(* Logix 5000 project; controller WWTP_SOLIDS_CLX vendor 1 type 14 code 54 rev 17.2; software revision 17.00; part 7 of 16 *)
(* tags used below, declared in another part *)
   Inp_PVBad : BOOL;   // 1=Scale PV or I/O Quality Bad, 0=OK
   Inp_PVUncertain : BOOL;   // 1=Scale PV Quality Uncertain, 0=OK
   Inp_CtrldEqpFault : BOOL;   // Controlled Equipment device or I/O status 0=OK, 1=fail
   Inp_Sim : BOOL;   // 1=Simulate working weigh scale; 0=use actual weight input
   Cfg_HasDribble : BOOL;   // 1=Slow to Dribble before complete, 0=use complete only
   Cfg_PCmdClear : BOOL;   // 1=Clear Program Commands on receipt 0=Leave Set
   Cfg_HasOverTolAlm : BOOL;   // 1=Over Tolerance Alarm exists and will be checked
   Cfg_HasUnderTolAlm : BOOL;   // 1=Under Tolerance Alarm exists and will be checked
   Cfg_HasTareFaultAlm : BOOL;   // 1=Tare Fault Alarm exists and will be checked
   Cfg_HasEqpFaultAlm : BOOL;   // 1=Equipment Fault Alarm exists and will be checked
   Cfg_OverTolResetReqd : BOOL;   // 1=Reset requied to clear Out of Tolerance High Alarm
   Cfg_UnderTolResetReqd : BOOL;   // 1=Reset required to clear Out of Tolerance Low Alarm
   Cfg_TareFaultResetReqd : BOOL;   // 1=Reset required to clear Tare Fault Alarm
   Cfg_EqpFaultResetReqd : BOOL;   // 1=Reset required to clear Equipment Fault Alarm
   Cfg_OverTolAckReqd : BOOL;   // 1=Acknowledge required for Out of Tolerance High Alarm
   Cfg_UnderTolAckReqd : BOOL;   // 1=Acknowledge required for Out of Tolerance Low Alarm
   Cfg_TareFaultAckReqd : BOOL;   // 1=Acknowledge required for Tare Fault Alarm
   Cfg_EqpFaultAckReqd : BOOL;   // 1=Acknowledge required for Equipment Fault Alarm
   Cfg_OverTolSeverity : SINT;   // Over Tolerance Alarm Severity 1=info, 2=warn, 3=excep, 4=fault
   Cfg_UnderTolSeverity : SINT;   // Under Tolerance Alarm Severity 1=info, 2=warn, 3=excep, 4=fault
   Cfg_TareFaultSeverity : SINT;   // Tare Fault Alarm Severity 1=info, 2=warn, 3=excep, 4=fault
   Cfg_EqpFaultSeverity : SINT;   // Equipment Fault Alarm Severity 1=info, 2=warn, 3=excep, 4=fault
   Cfg_InpRawMin : REAL;   // Minimum unscaled weight input
   Cfg_InpRawMax : REAL;   // Maximum unscaled weight input
   Cfg_PVEUMin : REAL;   // Minimum scaled weight PV input (EU)
   Cfg_PVEUMax : REAL;   // Maximum scaled weight PV input (EU)
   Cfg_MaxQty : REAL;   // Maximum allowed quantity to deliver (setpoint) (EU)
   Cfg_RateTime : REAL;   // Time factor for rate (60 for /min, 3600 for /hr) (Sec)
   Cfg_RateFiltTC : REAL;   // Filter Time Constant (sec) for calculated Rate
   Cfg_TareFaultLim : REAL;   // Amount (EU) scale can drift after Tare before starting flow without Faulting
   Cfg_SimStartWt : REAL;   // Weight to start from (tare to) in simulation (EU)
   Cfg_SimRate : REAL;   // Rate at which to deliver when running in Simulation (EU/rate time)
   Cfg_SimDribbleRate : REAL;   // Rate at which to dribble when running in Simulation (EU/rate time)
   PCmd_OverTolAck : BOOL;   // Program Command to Acknowledge Out of Tolerance High Alarm
   PCmd_OverTolInhibit : BOOL;   // Program Command to Inhibit Out of Tolerance High Alarm
   PCmd_OverTolUninhibit : BOOL;   // Program Command to Uninhibit Out of Tolerance High Alarm
   PCmd_UnderTolAck : BOOL;   // Program Command to Acknowledge Out of Tolerance Low Alarm
   PCmd_UnderTolInhibit : BOOL;   // Program Command to Inhibit Out of Tolerance Low Alarm
   PCmd_UnderTolUninhibit : BOOL;   // Program Command to Uninhibit Out of Tolerance Low Alarm
   PCmd_TareFaultAck : BOOL;   // Program Command to Acknowledge Tare Fault Alarm
   PCmd_TareFaultInhibit : BOOL;   // Program Command to Inhibit Tare Fault Alarm
   PCmd_TareFaultUninhibit : BOOL;   // Program Command to Uninhibit Tare Fault Alarm
   PCmd_EqpFaultAck : BOOL;   // Program Command to Acknowledge Equipment Fault Alarm
   PCmd_EqpFaultInhibit : BOOL;   // Program Command to Inhibit Equipment Fault Alarm
   PCmd_EqpFaultUninhibit : BOOL;   // Program Command to Uninhibit Equipment Fault Alarm
   Out_RunFlow : BOOL;   // 1=Deliver at Full (fast) Flow
   Out_DribbleFlow : BOOL;   // 1=Deliver at Dribble (slow) Flow
   Out_StopFlow : BOOL;   // 1=Stop Delivery Equipment
   Val_Qty : REAL;   // Quantity actually delivered (totalizer output) (EU)
   Val_SP : REAL;   // Amount to be delivered (Setpoint) (EU)
   Val_PctComplete : REAL;   // Percent Complete (for Progress Bar on HMI) 0.0 to 100.0%
   Val_DribbleQty : REAL;   // Amount to be delivered at slow rate (EU)
   Val_Preact : REAL;   // Amount before SP at which flow will be stopped (EU)
   Val_PVEUMin : REAL;   // Minimum of scaled range = MIN (Cfg_PVEUMin, Cfg_PVEUMax)
   Val_PVEUMax : REAL;   // Maximum of scaled range = MAX (Cfg_PVEUMin, Cfg_PVEUMax)
   Val_Notify : SINT;   // Current Alarm Level and Acknowledgement (enumeration)
   Sts_Tared : BOOL;   // Scale Tare completed, Qty = 0.0
   Sts_FlowRunning : BOOL;   // 1=Flow is Running (Out_Run is ON)
   Sts_FlowDribble : BOOL;   // 1=Flow is slowed to Dribble (Out_Dribble is ON)
   Sts_FlowStopped : BOOL;   // 1=Flow is Stopped (Out_Stop is ON)
   Sts_Bumping : BOOL;   // 1=Bump flow (timed) is active
   Sts_Complete : BOOL;   // 1=Total Delivered > (SP - Preact)
   Sts_Available : BOOL;   // 1=Dosing available for control by automation (Prog)
   Sts_PVBad : BOOL;   // 1=Weight PV and Rate PV Quality Bad (I/O fail), 0=OK
   Sts_PVUncertain : BOOL;   // 1=Weight PV and Rate PV Quality is Uncertian, 0=OK
   Sts_Err : BOOL;   // 1=Error: Bad Configuration, see detail Err bits for reason
   Err_Raw : BOOL;   // 1=Error: Cfg_InpRawMax or Cfg_InpRawMin invalid
   Err_EU : BOOL;   // 1=Error: Cfg_PVEUMax or Cfg_PVEUMin invalid
   Err_Rate : BOOL;   // 1=Error: Cfg_RateFiltTC or Cfg_RateTime invalid
   Err_Limit : BOOL;   // 1=Error: Cfg_MaxQty invalid
   Err_Sim : BOOL;   // 1=Error: Cfg_SimDribbleRate or Cfg_SimRate invalid
   Err_Timer : BOOL;   // 1=Error: Cfg_BumpT (use 0.0 to 2147483.647)
   Err_Alarm : BOOL;   // 1=Error: Alarm Min Duration or Severity Cfg Invalid
   Sts_Maint : BOOL;   // 1=Mode is Maintenance (supersedes Prog, Oper)
   Sts_Prog : BOOL;   // 1=Mode is Program (auto)
   Sts_Oper : BOOL;   // 1=Mode is Operator (manual)
   Sts_ProgOperLock : BOOL;   // 1=Program or Operator has requested Mode Lock
   Sts_OverTol : BOOL;   // 1=Delivery Out of Tolerance High
   Alm_OverTol : BOOL;   // 1=Delivery Out of Tolerance High Alarm
   Ack_OverTol : BOOL;   // 1=Out of Tolerance High Alarm has been acknowledged
   Sts_OverTolDisabled : BOOL;   // 1=Out of Tolerance High Alarm has been disabled (will not be sent)
   Sts_OverTolInhibited : BOOL;   // 1=Out of Tolerance High Alarm has been inhibited by logic
   Sts_OverTolSuppressed : BOOL;   // 1=Out of Tolerance High Alarm has been suppressed (logged only)
   Sts_UnderTol : BOOL;   // 1=Delivery Out of Tolerance Low
   Alm_UnderTol : BOOL;   // 1=Delivery Out of Tolerance Low Alarm
   Ack_UnderTol : BOOL;   // 1=Out of Tolerance Low Alarm has been acknowledged
   Sts_UnderTolDisabled : BOOL;   // 1=Out of Tolerance Low Alarm has been disabled (will not be sent)
   Sts_UnderTolInhibited : BOOL;   // 1=Out of Tolerance Low Alarm has been inhibited by logic
   Sts_UnderTolSuppressed : BOOL;   // 1=Out of Tolerance Low Alarm has been suppressed (logged only)
   Sts_TareFault : BOOL;   // 1=Scale reading moved unexpectedly since Tare
   Alm_TareFault : BOOL;   // 1=Warning: scale reading moved since Tare
   Ack_TareFault : BOOL;   // 1=Tare Fault Alarm has been acknowledged
   Sts_TareFaultDisabled : BOOL;   // 1=Tare Fault Alarm is Disabled (not saved or sent)
   Sts_TareFaultInhibited : BOOL;   // 1=Tare Fault Alarm has been inhibited by logic
   Sts_TareFaultSuppressed : BOOL;   // 1=Tare Fault Alarm has been suppressed (logged only)
   Sts_EqpFault : BOOL;   // 1=Equipment Fault Detected
   Alm_EqpFault : BOOL;   // 1=Equipment Fault Alarm
   Ack_EqpFault : BOOL;   // 1=Equipment Fault Alarm has been acknowledged
   Sts_EqpFaultDisabled : BOOL;   // 1=Equipment Fault Alarm is Disabled (not saved or sent)
   Sts_EqpFaultInhibited : BOOL;   // 1=Equipment Fault Alarm has been inhibited by logic
   Sts_EqpFaultSuppressed : BOOL;   // 1=Equipment Fault Alarm has been suppressed (logged only)
   Rdy_Tare : BOOL;   // 1=Ready for OCmd_Tare (enables button)
   Rdy_StartFlow : BOOL;   // 1=Ready for OCmd_StartFlow (enables button)
   Rdy_StopFlow : BOOL;   // 1=Ready for OCmd_StopFlow (enables button)
   Rdy_CheckTol : BOOL;   // 1-Ready for OCmd_CheckTol (enables button)
   Rdy_Bump : BOOL;   // 1=Ready for OCmd_Bump (enables button)
   Rdy_Reset : BOOL;   // 1=Ready for OCmd_Reset (enables button)
   Wrk_Notify : DINT;   // Buffer for building Val_Notify
   Mode : P_Mode;   // Analog Input Mode Selection
   Wrk_Tare : BOOL;   // Request to Tare Scale received
   TareFault : P_Alarm;   // Scale not holding at point at which Tared Alarm
   UnderTol : P_Alarm;   // Final Quantity Below Low Tolerance Alarm
   OverTol : P_Alarm;   // Final Quantity Above High Tolerance Alarm
   EqpFault : P_Alarm;   // Equipment (Sensor, Controlled Equip.) Fault Alarm
   Wrk_RunFlow : BOOL;   // 1=Flow (full)( should be running
   Wrk_BumpFlow : BOOL;   // Operator requested bump flow to make up Under Tolerance
   Wrk_BumpT : TIMER;   // Bump Timer for shot of flow to make up Under Tolerance
   Wrk_PctComplete : REAL;   // Percent Complete calculation intermediate
   Wrk_InpInfNaN : BOOL;   // Input Weight is Infinite or NaN
(* P_DoseWS, continued *)

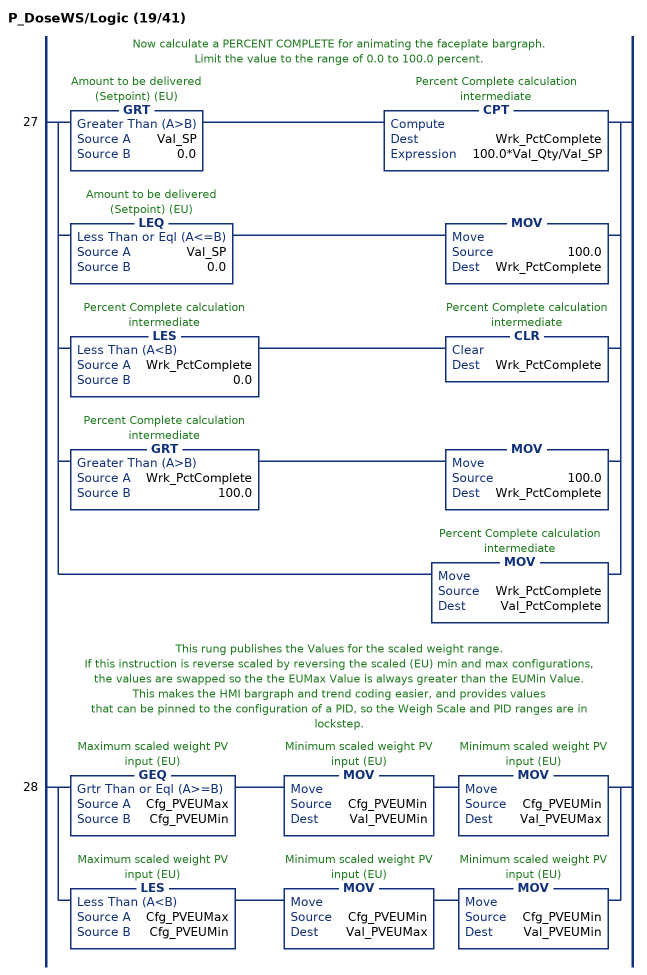
   [picture p136: P_DoseWS/Logic rungs 27-28]
   // Now calculate a PERCENT COMPLETE for animating the faceplate bargraph.
   // Limit the value to the range of 0.0 to 100.0 percent.
   27: [GRT(Val_SP,0.0) CPT(Wrk_PctComplete,100.0*Val_Qty/Val_SP) ,LEQ(Val_SP,0.0) MOV(100.0,Wrk_PctComplete) ,LES(Wrk_PctComplete,0.0) CLR(Wrk_PctComplete) ,GRT(Wrk_PctComplete,100.0) MOV(100.0,Wrk_PctComplete) ,MOV(Wrk_PctComplete,Val_PctComplete) ];
   // This rung publishes the Values for the scaled weight range.
   // If this instruction is reverse scaled by reversing the scaled (EU) min and max configurations,
   // the values are swapped so the the EUMax Value is always greater than the EUMin Value.
   // This makes the HMI bargraph and trend coding easier, and provides values
   // that can be pinned to the configuration of a PID, so the Weigh Scale and PID ranges are in lockstep.
   28: [GEQ(Cfg_PVEUMax,Cfg_PVEUMin) MOV(Cfg_PVEUMin,Val_PVEUMin) MOV(Cfg_PVEUMin,Val_PVEUMax) ,LES(Cfg_PVEUMax,Cfg_PVEUMin) MOV(Cfg_PVEUMin,Val_PVEUMax) MOV(Cfg_PVEUMin,Val_PVEUMin) ];
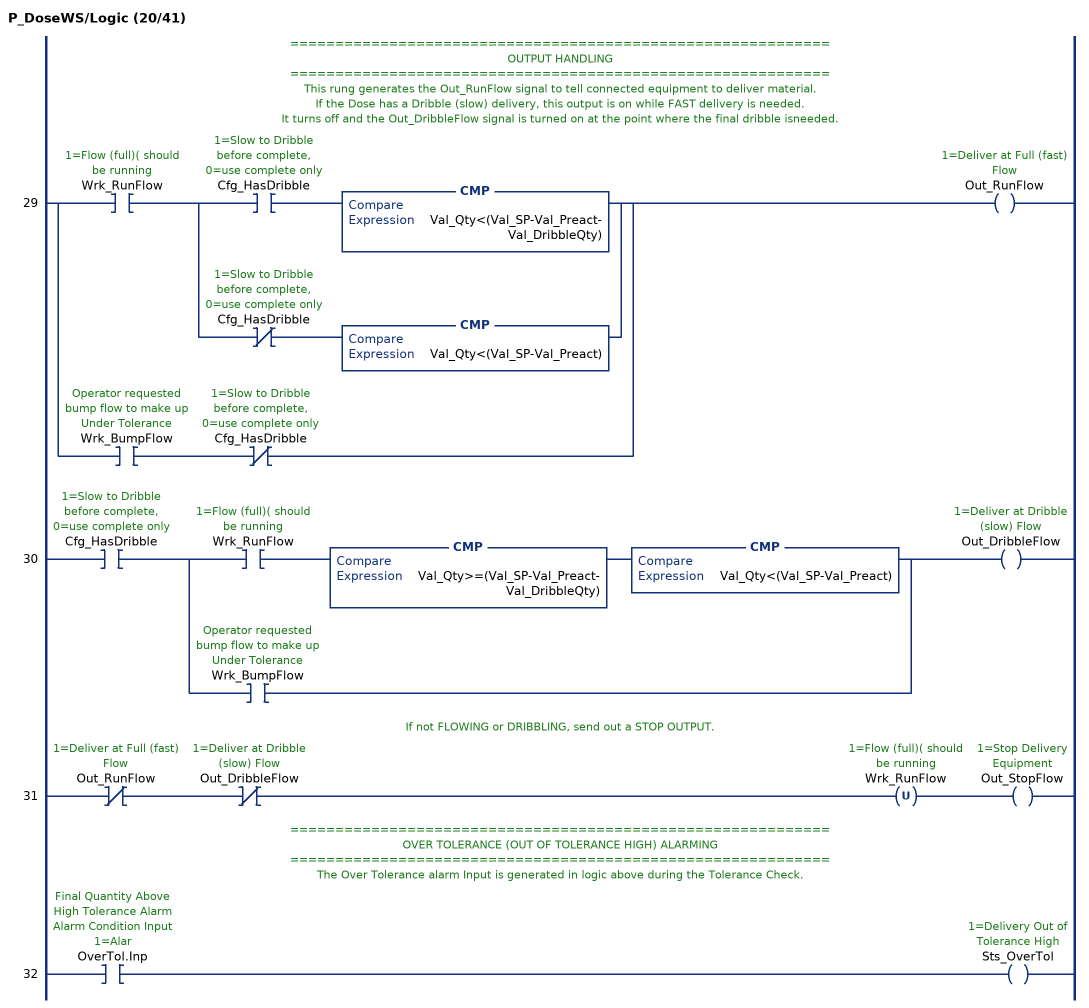
   // ============================================================
   // OUTPUT HANDLING
   // ============================================================
   // This rung generates the Out_RunFlow signal to tell connected equipment to deliver material.
   // If the Dose has a Dribble (slow) delivery, this output is on while FAST delivery is needed.
   // It turns off and the Out_DribbleFlow signal is turned on at the point where the final dribble isneeded.
   29: [XIC(Wrk_RunFlow) [XIC(Cfg_HasDribble) CMP(Val_Qty<(Val_SP-Val_Preact-Val_DribbleQty)) ,XIO(Cfg_HasDribble) CMP(Val_Qty<(Val_SP-Val_Preact)) ] ,XIC(Wrk_BumpFlow) XIO(Cfg_HasDribble) ]OTE(Out_RunFlow);
   30: XIC(Cfg_HasDribble)[XIC(Wrk_RunFlow) CMP(Val_Qty>=(Val_SP-Val_Preact-Val_DribbleQty)) CMP(Val_Qty<(Val_SP-Val_Preact)) ,XIC(Wrk_BumpFlow) ]OTE(Out_DribbleFlow);
   // If not FLOWING or DRIBBLING, send out a STOP OUTPUT.
   31: XIO(Out_RunFlow)XIO(Out_DribbleFlow)OTU(Wrk_RunFlow)OTE(Out_StopFlow);
   // ============================================================
   // OVER TOLERANCE (OUT OF TOLERANCE HIGH) ALARMING
   // ============================================================
   // The Over Tolerance alarm Input is generated in logic above during the Tolerance Check.
   32: XIC(OverTol.Inp)OTE(Sts_OverTol);
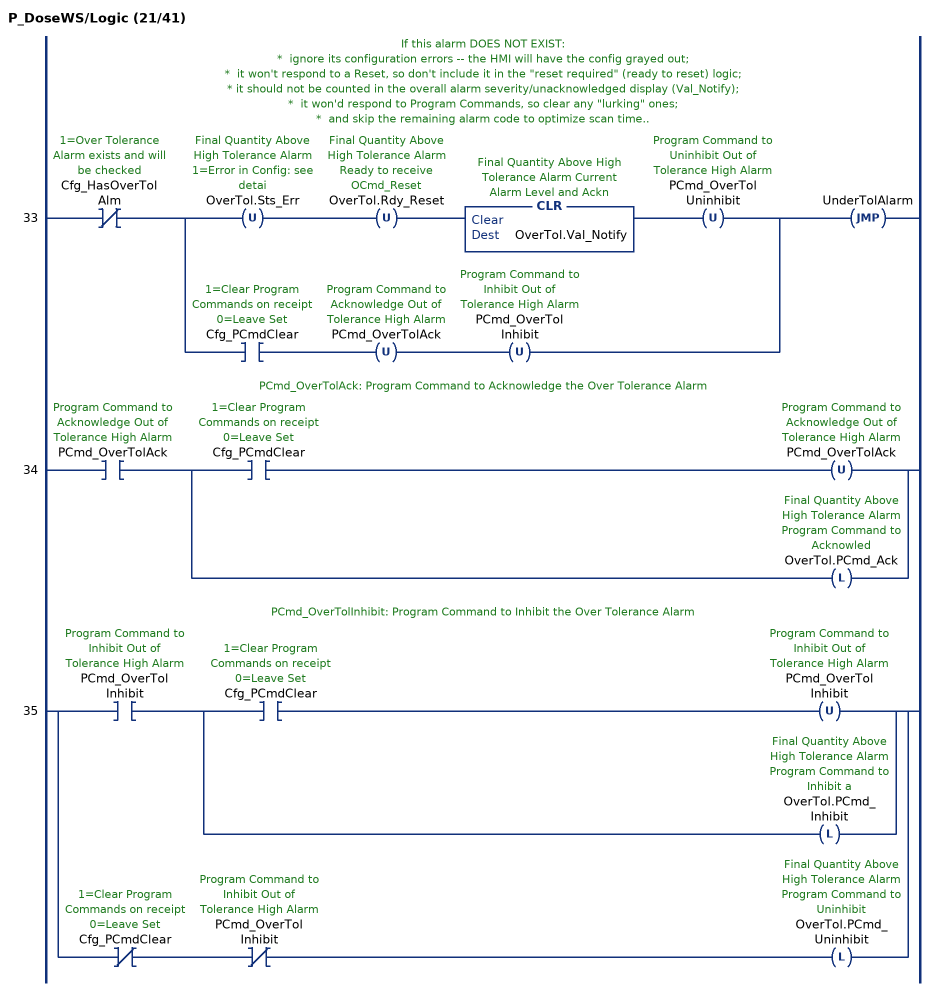
   // If this alarm DOES NOT EXIST:
   // *  ignore its configuration errors -- the HMI will have the config grayed out;
   // *  it won't respond to a Reset, so don't include it in the "reset required" (ready to reset) logic;
   // * it should not be counted in the overall alarm severity/unacknowledged display (Val_Notify);
   // *  it won'd respond to Program Commands, so clear any "lurking" ones;
   // *  and skip the remaining alarm code to optimize scan time..
   33: XIO(Cfg_HasOverTolAlm)[OTU(OverTol.Sts_Err) OTU(OverTol.Rdy_Reset) CLR(OverTol.Val_Notify) OTU(PCmd_OverTolUninhibit) ,XIC(Cfg_PCmdClear) OTU(PCmd_OverTolAck) OTU(PCmd_OverTolInhibit) ]JMP(UnderTolAlarm);
   // PCmd_OverTolAck: Program Command to Acknowledge the Over Tolerance Alarm
   34: XIC(PCmd_OverTolAck)[XIC(Cfg_PCmdClear) OTU(PCmd_OverTolAck) ,OTL(OverTol.PCmd_Ack) ];
   // PCmd_OverTolInhibit: Program Command to Inhibit the Over Tolerance Alarm
   35: [XIC(PCmd_OverTolInhibit) [XIC(Cfg_PCmdClear) OTU(PCmd_OverTolInhibit) ,OTL(OverTol.PCmd_Inhibit) ] ,XIO(Cfg_PCmdClear) XIO(PCmd_OverTolInhibit) OTL(OverTol.PCmd_Uninhibit) ];
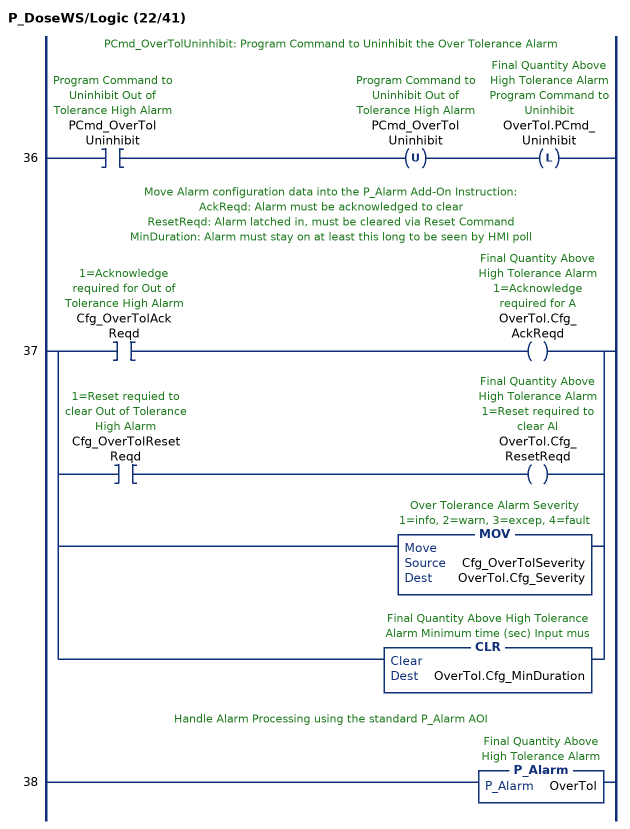
   // PCmd_OverTolUninhibit: Program Command to Uninhibit the Over Tolerance Alarm
   36: XIC(PCmd_OverTolUninhibit)OTU(PCmd_OverTolUninhibit)OTL(OverTol.PCmd_Uninhibit);
   // Move Alarm configuration data into the P_Alarm Add-On Instruction:
   // AckReqd: Alarm must be acknowledged to clear
   // ResetReqd: Alarm latched in, must be cleared via Reset Command
   // MinDuration: Alarm must stay on at least this long to be seen by HMI poll
   37: [XIC(Cfg_OverTolAckReqd) OTE(OverTol.Cfg_AckReqd) ,XIC(Cfg_OverTolResetReqd) OTE(OverTol.Cfg_ResetReqd) ,MOV(Cfg_OverTolSeverity,OverTol.Cfg_Severity) ,CLR(OverTol.Cfg_MinDuration) ];
   // Handle Alarm Processing using the standard P_Alarm AOI
   38: P_Alarm(OverTol);
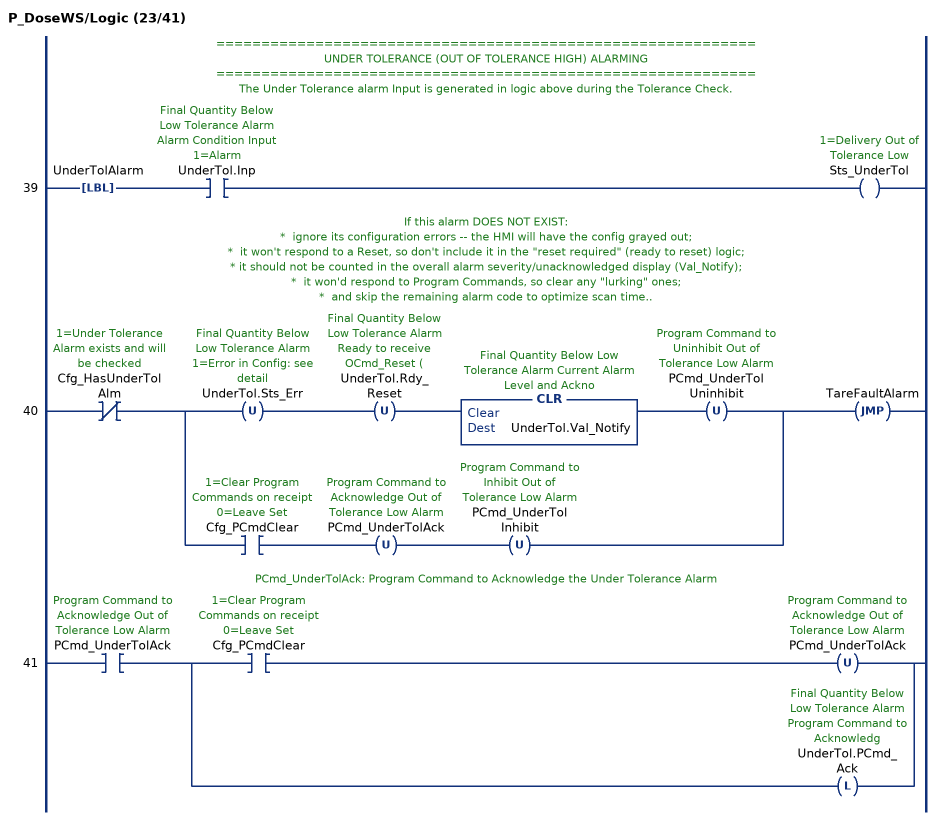
   // ============================================================
   // UNDER TOLERANCE (OUT OF TOLERANCE HIGH) ALARMING
   // ============================================================
   // The Under Tolerance alarm Input is generated in logic above during the Tolerance Check.
   39: LBL(UnderTolAlarm)XIC(UnderTol.Inp)OTE(Sts_UnderTol);
   // If this alarm DOES NOT EXIST:
   // *  ignore its configuration errors -- the HMI will have the config grayed out;
   // *  it won't respond to a Reset, so don't include it in the "reset required" (ready to reset) logic;
   // * it should not be counted in the overall alarm severity/unacknowledged display (Val_Notify);
   // *  it won'd respond to Program Commands, so clear any "lurking" ones;
   // *  and skip the remaining alarm code to optimize scan time..
   40: XIO(Cfg_HasUnderTolAlm)[OTU(UnderTol.Sts_Err) OTU(UnderTol.Rdy_Reset) CLR(UnderTol.Val_Notify) OTU(PCmd_UnderTolUninhibit) ,XIC(Cfg_PCmdClear) OTU(PCmd_UnderTolAck) OTU(PCmd_UnderTolInhibit) ]JMP(TareFaultAlarm);
   // PCmd_UnderTolAck: Program Command to Acknowledge the Under Tolerance Alarm
   41: XIC(PCmd_UnderTolAck)[XIC(Cfg_PCmdClear) OTU(PCmd_UnderTolAck) ,OTL(UnderTol.PCmd_Ack) ];
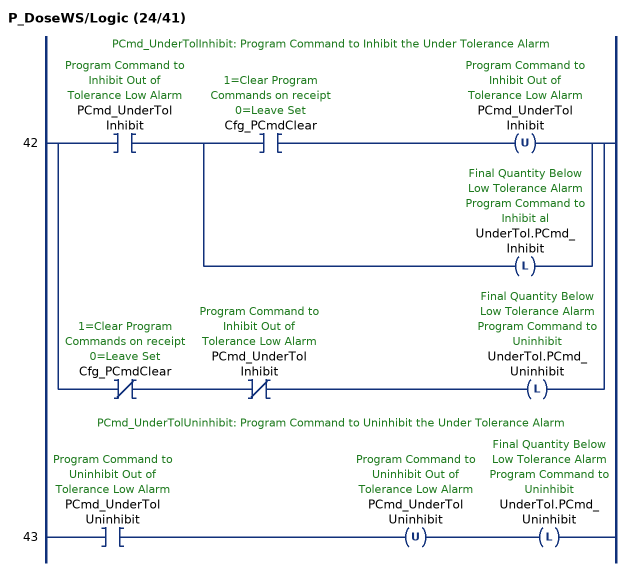
   // PCmd_UnderTolInhibit: Program Command to Inhibit the Under Tolerance Alarm
   42: [XIC(PCmd_UnderTolInhibit) [XIC(Cfg_PCmdClear) OTU(PCmd_UnderTolInhibit) ,OTL(UnderTol.PCmd_Inhibit) ] ,XIO(Cfg_PCmdClear) XIO(PCmd_UnderTolInhibit) OTL(UnderTol.PCmd_Uninhibit) ];
   // PCmd_UnderTolUninhibit: Program Command to Uninhibit the Under Tolerance Alarm
   43: XIC(PCmd_UnderTolUninhibit)OTU(PCmd_UnderTolUninhibit)OTL(UnderTol.PCmd_Uninhibit);
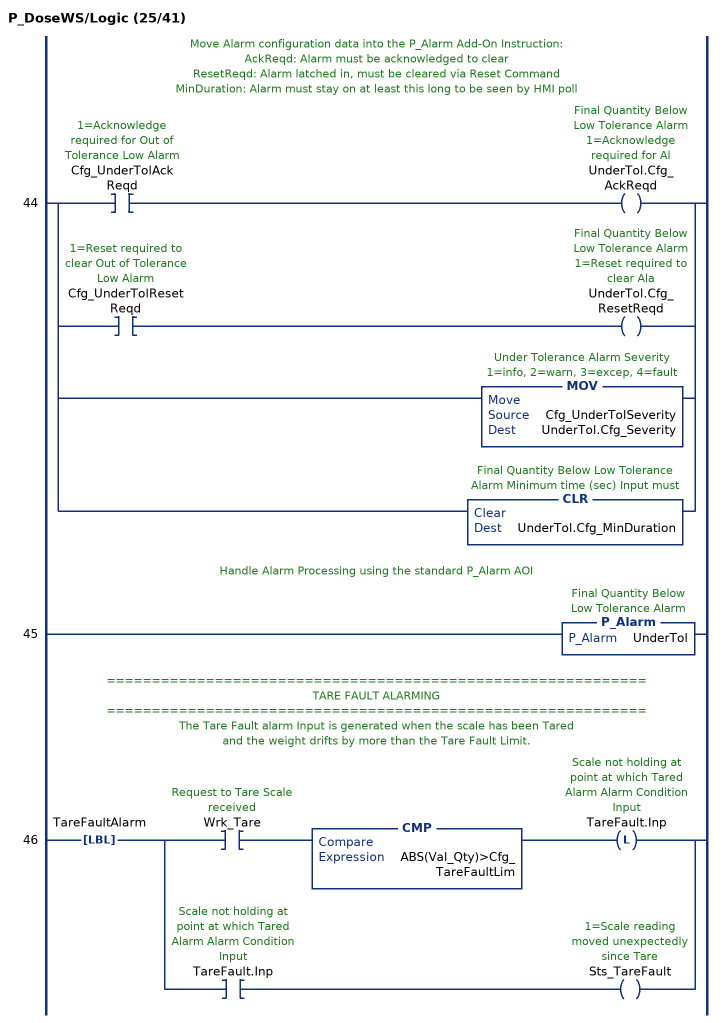
   // Move Alarm configuration data into the P_Alarm Add-On Instruction:
   // AckReqd: Alarm must be acknowledged to clear
   // ResetReqd: Alarm latched in, must be cleared via Reset Command
   // MinDuration: Alarm must stay on at least this long to be seen by HMI poll
   44: [XIC(Cfg_UnderTolAckReqd) OTE(UnderTol.Cfg_AckReqd) ,XIC(Cfg_UnderTolResetReqd) OTE(UnderTol.Cfg_ResetReqd) ,MOV(Cfg_UnderTolSeverity,UnderTol.Cfg_Severity) ,CLR(UnderTol.Cfg_MinDuration) ];
   // Handle Alarm Processing using the standard P_Alarm AOI
   45: P_Alarm(UnderTol);
   // ============================================================
   // TARE FAULT ALARMING
   // ============================================================
   // The Tare Fault alarm Input is generated when the scale has been Tared
   // and the weight drifts by more than the Tare Fault Limit.
   46: LBL(TareFaultAlarm)[XIC(Wrk_Tare) CMP(ABS(Val_Qty)>Cfg_TareFaultLim) OTL(TareFault.Inp) ,XIC(TareFault.Inp) OTE(Sts_TareFault) ];
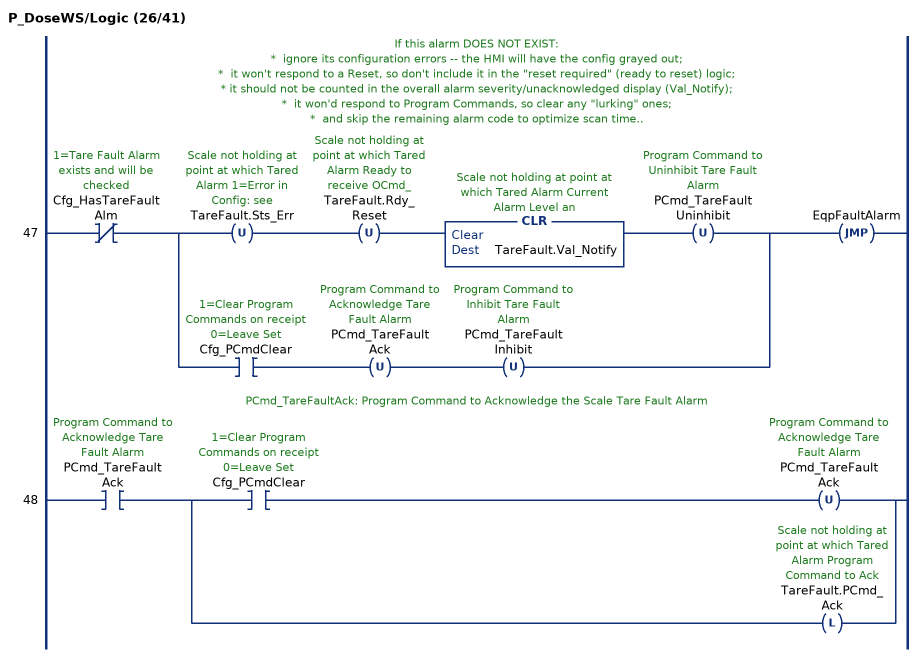
   // If this alarm DOES NOT EXIST:
   // *  ignore its configuration errors -- the HMI will have the config grayed out;
   // *  it won't respond to a Reset, so don't include it in the "reset required" (ready to reset) logic;
   // * it should not be counted in the overall alarm severity/unacknowledged display (Val_Notify);
   // *  it won'd respond to Program Commands, so clear any "lurking" ones;
   // *  and skip the remaining alarm code to optimize scan time..
   47: XIO(Cfg_HasTareFaultAlm)[OTU(TareFault.Sts_Err) OTU(TareFault.Rdy_Reset) CLR(TareFault.Val_Notify) OTU(PCmd_TareFaultUninhibit) ,XIC(Cfg_PCmdClear) OTU(PCmd_TareFaultAck) OTU(PCmd_TareFaultInhibit) ]JMP(EqpFaultAlarm);
   // PCmd_TareFaultAck: Program Command to Acknowledge the Scale Tare Fault Alarm
   48: XIC(PCmd_TareFaultAck)[XIC(Cfg_PCmdClear) OTU(PCmd_TareFaultAck) ,OTL(TareFault.PCmd_Ack) ];
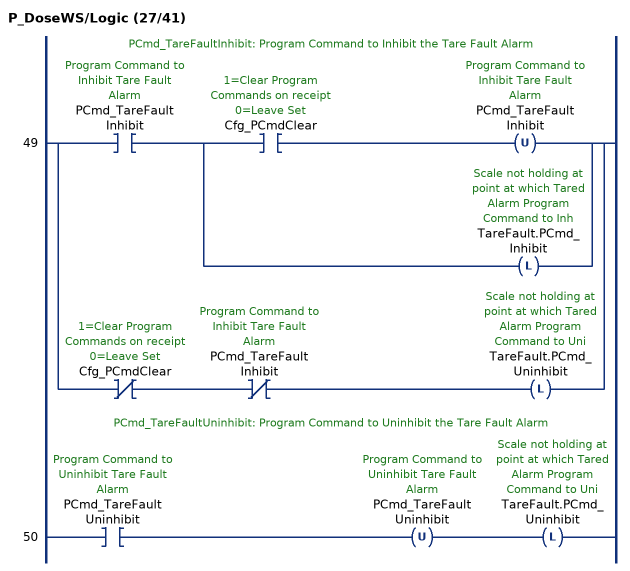
   // PCmd_TareFaultInhibit: Program Command to Inhibit the Tare Fault Alarm
   49: [XIC(PCmd_TareFaultInhibit) [XIC(Cfg_PCmdClear) OTU(PCmd_TareFaultInhibit) ,OTL(TareFault.PCmd_Inhibit) ] ,XIO(Cfg_PCmdClear) XIO(PCmd_TareFaultInhibit) OTL(TareFault.PCmd_Uninhibit) ];
   // PCmd_TareFaultUninhibit: Program Command to Uninhibit the Tare Fault Alarm
   50: XIC(PCmd_TareFaultUninhibit)OTU(PCmd_TareFaultUninhibit)OTL(TareFault.PCmd_Uninhibit);
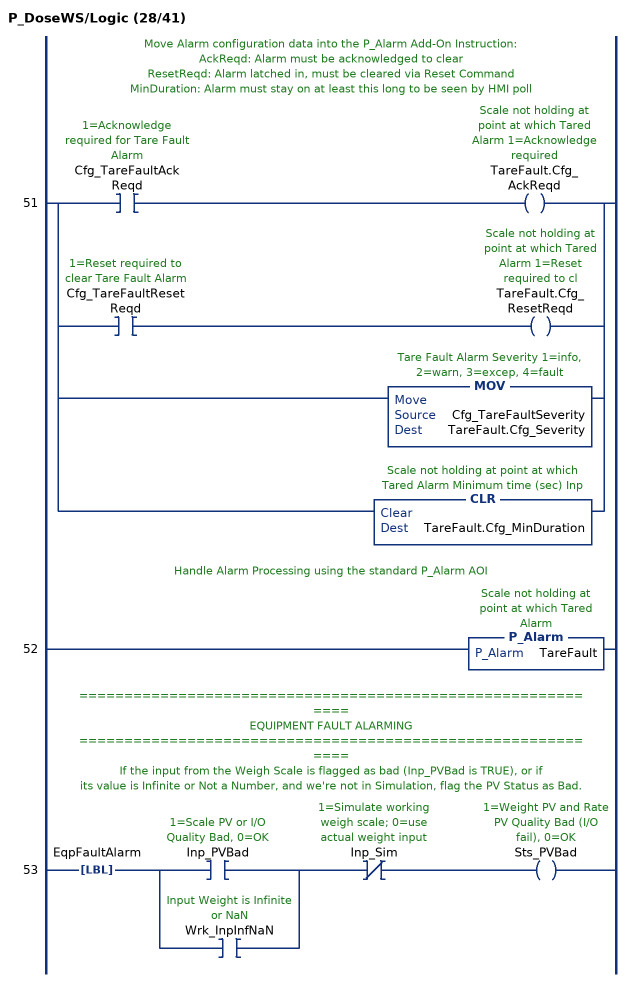
   // Move Alarm configuration data into the P_Alarm Add-On Instruction:
   // AckReqd: Alarm must be acknowledged to clear
   // ResetReqd: Alarm latched in, must be cleared via Reset Command
   // MinDuration: Alarm must stay on at least this long to be seen by HMI poll
   51: [XIC(Cfg_TareFaultAckReqd) OTE(TareFault.Cfg_AckReqd) ,XIC(Cfg_TareFaultResetReqd) OTE(TareFault.Cfg_ResetReqd) ,MOV(Cfg_TareFaultSeverity,TareFault.Cfg_Severity) ,CLR(TareFault.Cfg_MinDuration) ];
   // Handle Alarm Processing using the standard P_Alarm AOI
   52: P_Alarm(TareFault);
   // ============================================================
   // EQUIPMENT FAULT ALARMING
   // ============================================================
   // If the input from the Weigh Scale is flagged as bad (Inp_PVBad is TRUE), or if
   // its value is Infinite or Not a Number, and we're not in Simulation, flag the PV Status as Bad.
   53: LBL(EqpFaultAlarm)[XIC(Inp_PVBad) ,XIC(Wrk_InpInfNaN) ]XIO(Inp_Sim)OTE(Sts_PVBad);
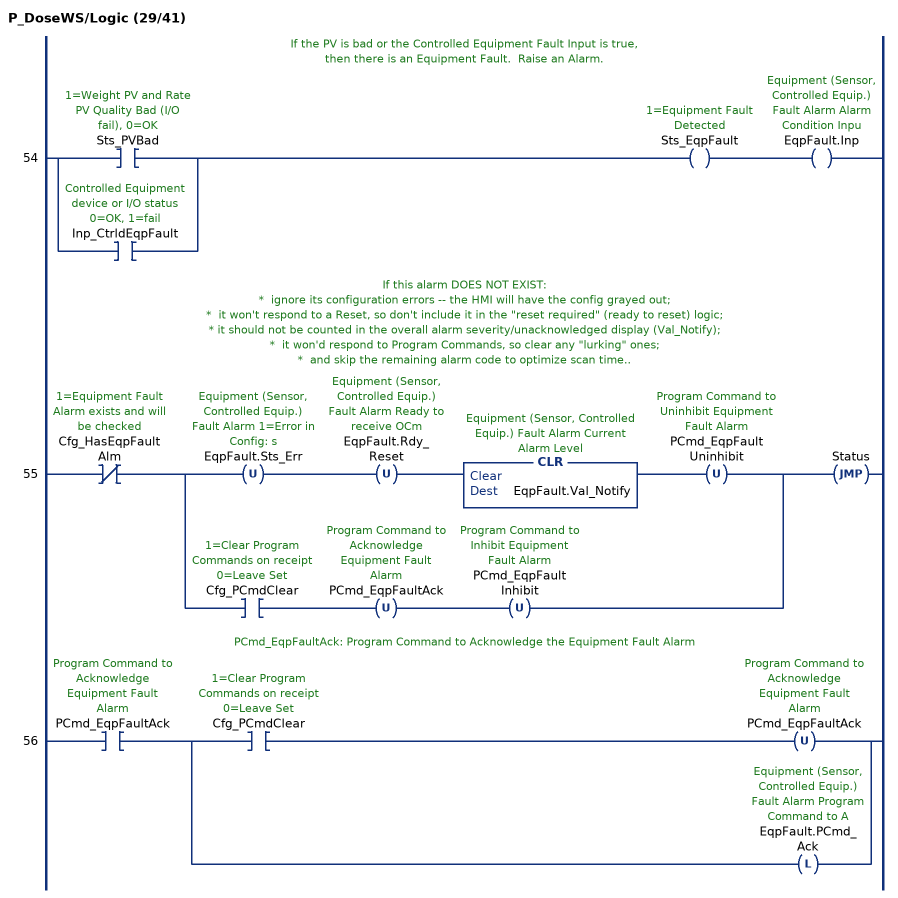
   // If the PV is bad or the Controlled Equipment Fault Input is true,
   // then there is an Equipment Fault.  Raise an Alarm.
   54: [XIC(Sts_PVBad) ,XIC(Inp_CtrldEqpFault) ]OTE(Sts_EqpFault)OTE(EqpFault.Inp);
   // If this alarm DOES NOT EXIST:
   // *  ignore its configuration errors -- the HMI will have the config grayed out;
   // *  it won't respond to a Reset, so don't include it in the "reset required" (ready to reset) logic;
   // * it should not be counted in the overall alarm severity/unacknowledged display (Val_Notify);
   // *  it won'd respond to Program Commands, so clear any "lurking" ones;
   // *  and skip the remaining alarm code to optimize scan time..
   55: XIO(Cfg_HasEqpFaultAlm)[OTU(EqpFault.Sts_Err) OTU(EqpFault.Rdy_Reset) CLR(EqpFault.Val_Notify) OTU(PCmd_EqpFaultUninhibit) ,XIC(Cfg_PCmdClear) OTU(PCmd_EqpFaultAck) OTU(PCmd_EqpFaultInhibit) ]JMP(Status);
   // PCmd_EqpFaultAck: Program Command to Acknowledge the Equipment Fault Alarm
   56: XIC(PCmd_EqpFaultAck)[XIC(Cfg_PCmdClear) OTU(PCmd_EqpFaultAck) ,OTL(EqpFault.PCmd_Ack) ];
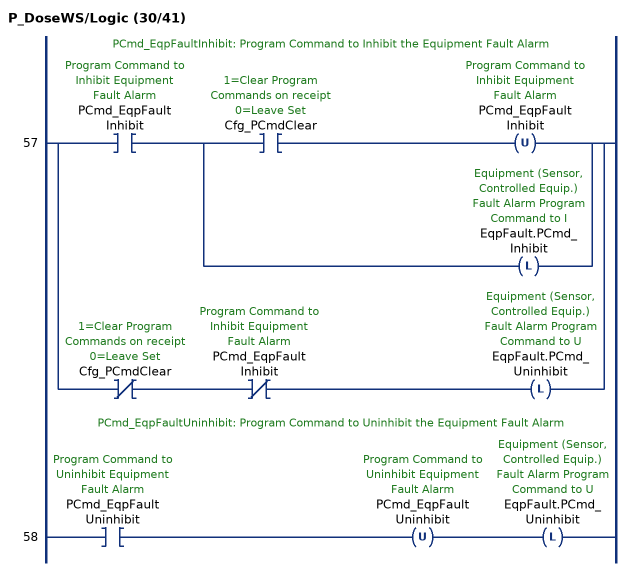
   // PCmd_EqpFaultInhibit: Program Command to Inhibit the Equipment Fault Alarm
   57: [XIC(PCmd_EqpFaultInhibit) [XIC(Cfg_PCmdClear) OTU(PCmd_EqpFaultInhibit) ,OTL(EqpFault.PCmd_Inhibit) ] ,XIO(Cfg_PCmdClear) XIO(PCmd_EqpFaultInhibit) OTL(EqpFault.PCmd_Uninhibit) ];
   // PCmd_EqpFaultUninhibit: Program Command to Uninhibit the Equipment Fault Alarm
   58: XIC(PCmd_EqpFaultUninhibit)OTU(PCmd_EqpFaultUninhibit)OTL(EqpFault.PCmd_Uninhibit);
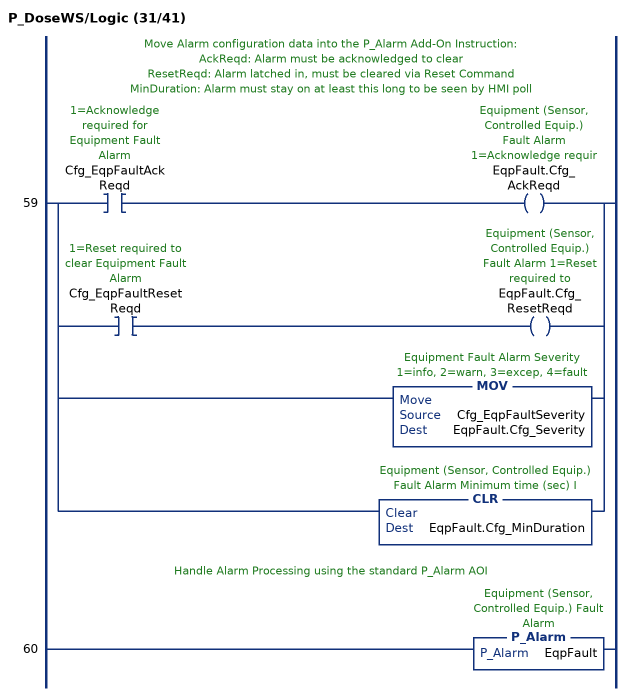
   // Move Alarm configuration data into the P_Alarm Add-On Instruction:
   // AckReqd: Alarm must be acknowledged to clear
   // ResetReqd: Alarm latched in, must be cleared via Reset Command
   // MinDuration: Alarm must stay on at least this long to be seen by HMI poll
   59: [XIC(Cfg_EqpFaultAckReqd) OTE(EqpFault.Cfg_AckReqd) ,XIC(Cfg_EqpFaultResetReqd) OTE(EqpFault.Cfg_ResetReqd) ,MOV(Cfg_EqpFaultSeverity,EqpFault.Cfg_Severity) ,CLR(EqpFault.Cfg_MinDuration) ];
   // Handle Alarm Processing using the standard P_Alarm AOI
   60: P_Alarm(EqpFault);
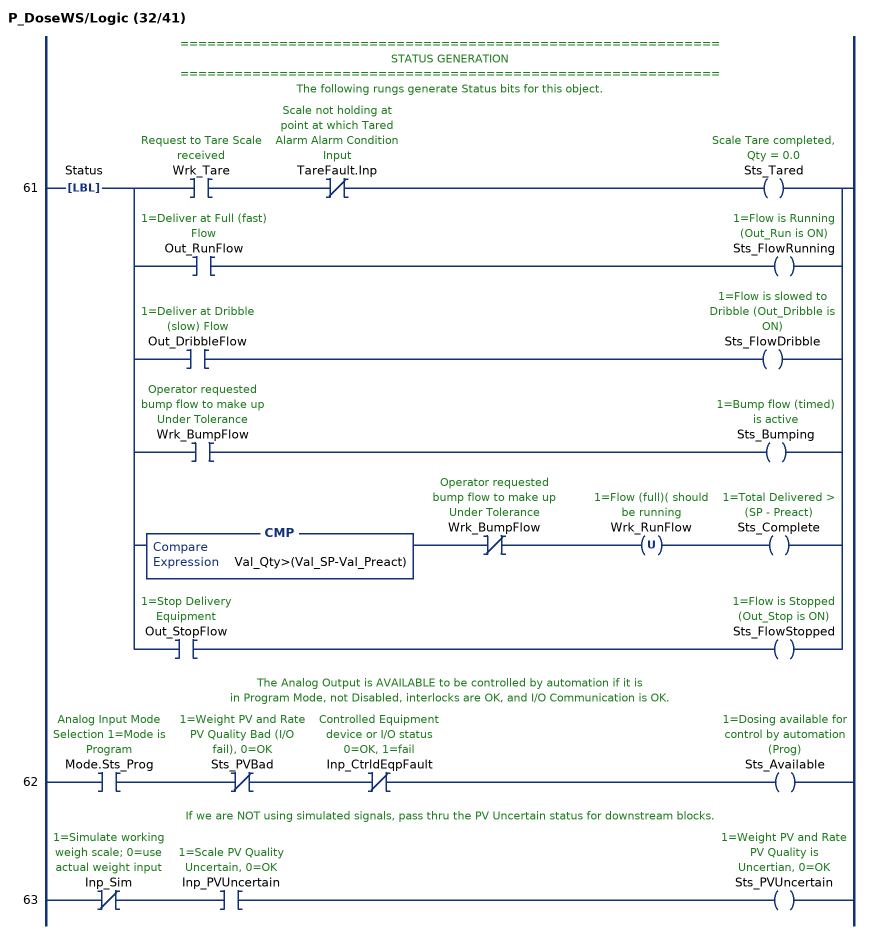
   // ============================================================
   // STATUS GENERATION
   // ============================================================
   // The following rungs generate Status bits for this object.
   61: LBL(Status)[XIC(Wrk_Tare) XIO(TareFault.Inp) OTE(Sts_Tared) ,XIC(Out_RunFlow) OTE(Sts_FlowRunning) ,XIC(Out_DribbleFlow) OTE(Sts_FlowDribble) ,XIC(Wrk_BumpFlow) OTE(Sts_Bumping) ,CMP(Val_Qty>(Val_SP-Val_Preact)) XIO(Wrk_BumpFlow) OTU(Wrk_RunFlow) OTE(Sts_Complete) ,XIC(Out_StopFlow) OTE(Sts_FlowStopped) ];
   // The Analog Output is AVAILABLE to be controlled by automation if it is
   // in Program Mode, not Disabled, interlocks are OK, and I/O Communication is OK.
   62: XIC(Mode.Sts_Prog)XIO(Sts_PVBad)XIO(Inp_CtrldEqpFault)OTE(Sts_Available);
   // If we are NOT using simulated signals, pass thru the PV Uncertain status for downstream blocks.
   63: XIO(Inp_Sim)XIC(Inp_PVUncertain)OTE(Sts_PVUncertain);
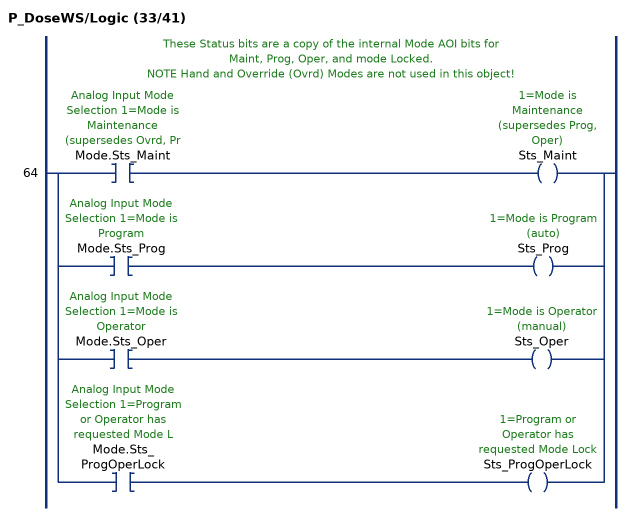
   // These Status bits are a copy of the internal Mode AOI bits for
   // Maint, Prog, Oper, and mode Locked.
   // NOTE Hand and Override (Ovrd) Modes are not used in this object!
   64: [XIC(Mode.Sts_Maint) OTE(Sts_Maint) ,XIC(Mode.Sts_Prog) OTE(Sts_Prog) ,XIC(Mode.Sts_Oper) OTE(Sts_Oper) ,XIC(Mode.Sts_ProgOperLock) OTE(Sts_ProgOperLock) ];
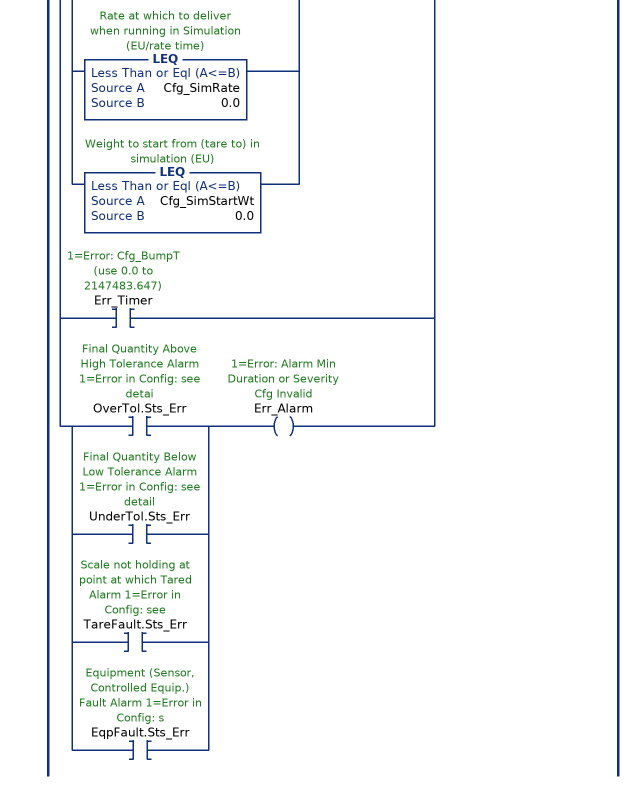
   // This rung handles the reports of all Error (Bad Configuration) Status.
   // Individual bits are provided for various status:
   // Invalid Raw (Unscaled) Units Scaling configs
   // Invalid Engineering Units Scaling configs
   // Invalid Rate calculation configs
   // Invalid Limit configs
   // Invalid Simulation configs
   // Invalid Timer configs (determined in Configuration section above)
   // Then a summary Error Status is provided, simply an OR of the individual bits.
   65: [EQU(Cfg_InpRawMax,Cfg_InpRawMin) OTE(Err_Raw) ,EQU(Cfg_PVEUMax,Cfg_PVEUMin) OTE(Err_EU) ,[LES(Cfg_RateFiltTC,0.0) ,LEQ(Cfg_RateTime,0.0) ] OTE(Err_Rate) ,[LEQ(Cfg_MaxQty,0.0) ,LES(Cfg_TareFaultLim,0.0) ] OTE(Err_Limit) ,[LEQ(Cfg_SimDribbleRate,0.0) ,LEQ(Cfg_SimRate,0.0) ,LEQ(Cfg_SimStartWt,0.0) ] OTE(Err_Sim) ,XIC(Err_Timer) ,[XIC(OverTol.Sts_Err) ,XIC(UnderTol.Sts_Err) ,XIC(TareFault.Sts_Err) ,XIC(EqpFault.Sts_Err) ] OTE(Err_Alarm) ]OTE(Sts_Err);
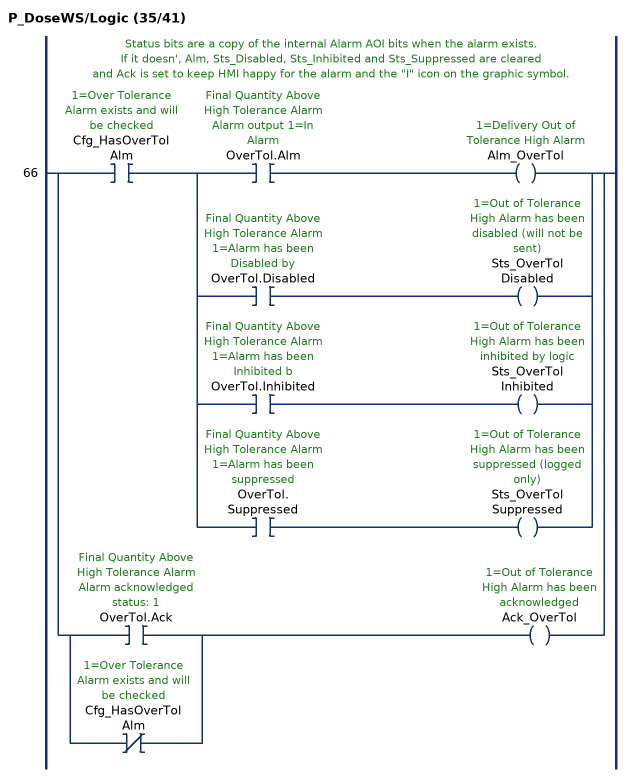
   // Status bits are a copy of the internal Alarm AOI bits when the alarm exists.
   // If it doesn', Alm, Sts_Disabled, Sts_Inhibited and Sts_Suppressed are cleared
   // and Ack is set to keep HMI happy for the alarm and the "I" icon on the graphic symbol.
   66: [XIC(Cfg_HasOverTolAlm) [XIC(OverTol.Alm) OTE(Alm_OverTol) ,XIC(OverTol.Disabled) OTE(Sts_OverTolDisabled) ,XIC(OverTol.Inhibited) OTE(Sts_OverTolInhibited) ,XIC(OverTol.Suppressed) OTE(Sts_OverTolSuppressed) ] ,[XIC(OverTol.Ack) ,XIO(Cfg_HasOverTolAlm) ] OTE(Ack_OverTol) ];
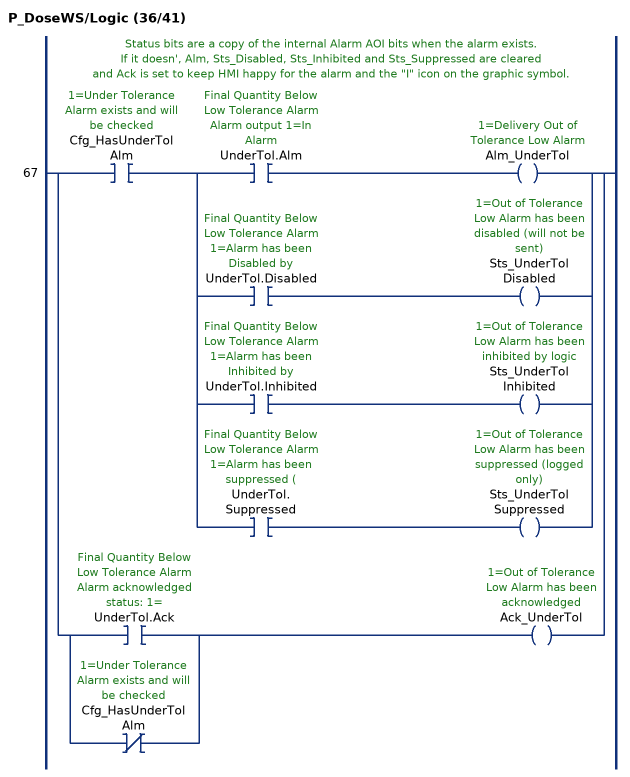
   // Status bits are a copy of the internal Alarm AOI bits when the alarm exists.
   // If it doesn', Alm, Sts_Disabled, Sts_Inhibited and Sts_Suppressed are cleared
   // and Ack is set to keep HMI happy for the alarm and the "I" icon on the graphic symbol.
   67: [XIC(Cfg_HasUnderTolAlm) [XIC(UnderTol.Alm) OTE(Alm_UnderTol) ,XIC(UnderTol.Disabled) OTE(Sts_UnderTolDisabled) ,XIC(UnderTol.Inhibited) OTE(Sts_UnderTolInhibited) ,XIC(UnderTol.Suppressed) OTE(Sts_UnderTolSuppressed) ] ,[XIC(UnderTol.Ack) ,XIO(Cfg_HasUnderTolAlm) ] OTE(Ack_UnderTol) ];
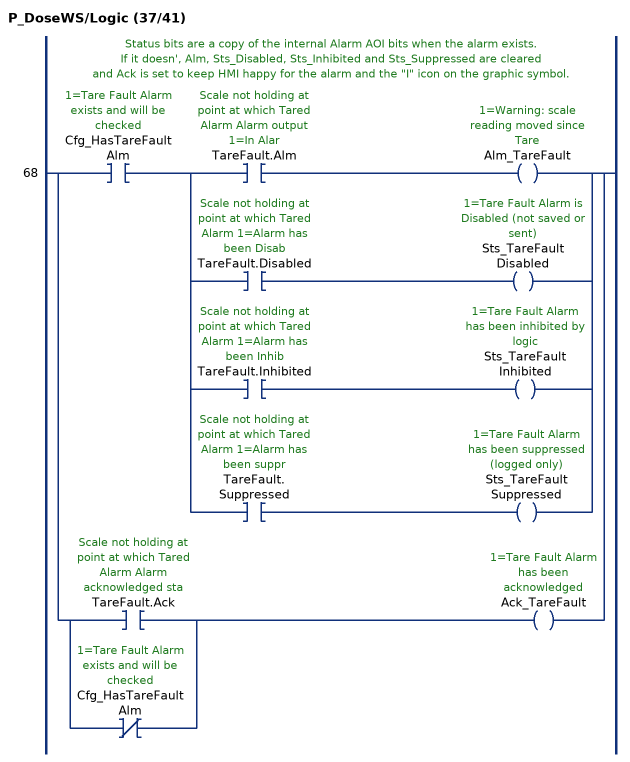
   // Status bits are a copy of the internal Alarm AOI bits when the alarm exists.
   // If it doesn', Alm, Sts_Disabled, Sts_Inhibited and Sts_Suppressed are cleared
   // and Ack is set to keep HMI happy for the alarm and the "I" icon on the graphic symbol.
   68: [XIC(Cfg_HasTareFaultAlm) [XIC(TareFault.Alm) OTE(Alm_TareFault) ,XIC(TareFault.Disabled) OTE(Sts_TareFaultDisabled) ,XIC(TareFault.Inhibited) OTE(Sts_TareFaultInhibited) ,XIC(TareFault.Suppressed) OTE(Sts_TareFaultSuppressed) ] ,[XIC(TareFault.Ack) ,XIO(Cfg_HasTareFaultAlm) ] OTE(Ack_TareFault) ];
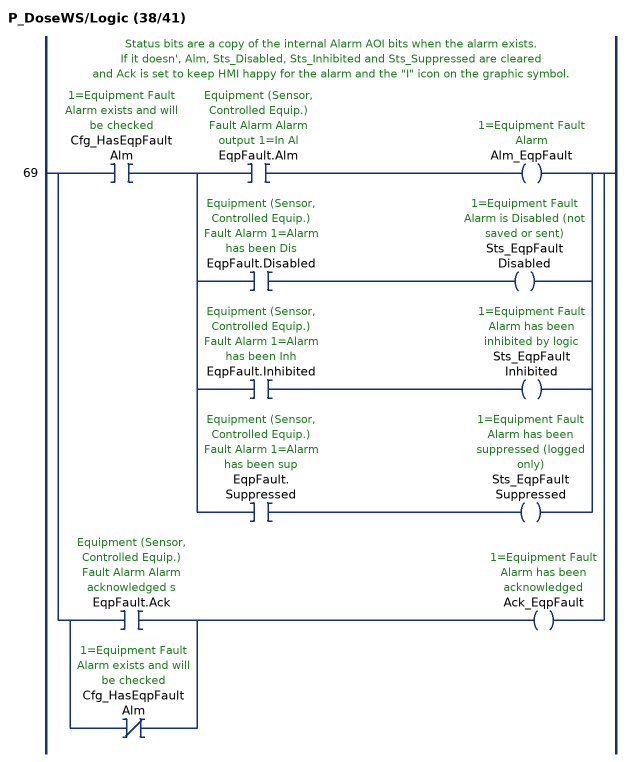
   // Status bits are a copy of the internal Alarm AOI bits when the alarm exists.
   // If it doesn', Alm, Sts_Disabled, Sts_Inhibited and Sts_Suppressed are cleared
   // and Ack is set to keep HMI happy for the alarm and the "I" icon on the graphic symbol.
   69: [XIC(Cfg_HasEqpFaultAlm) [XIC(EqpFault.Alm) OTE(Alm_EqpFault) ,XIC(EqpFault.Disabled) OTE(Sts_EqpFaultDisabled) ,XIC(EqpFault.Inhibited) OTE(Sts_EqpFaultInhibited) ,XIC(EqpFault.Suppressed) OTE(Sts_EqpFaultSuppressed) ] ,[XIC(EqpFault.Ack) ,XIO(Cfg_HasEqpFaultAlm) ] OTE(Ack_EqpFault) ];
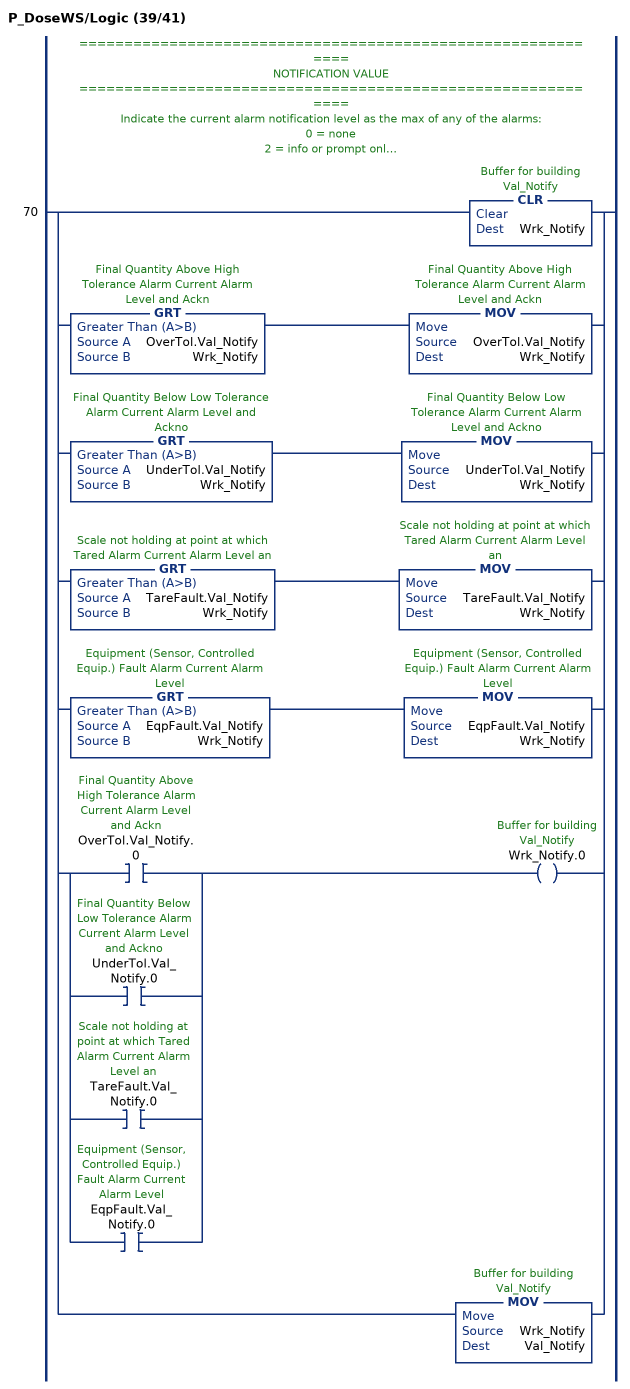
   // ============================================================
   // NOTIFICATION VALUE
   // ============================================================
   // Indicate the current alarm notification level as the max of any of the alarms:
   // 0 = none
   // 2 = info or prompt only
   // 4 = warning
   // 6 = exception (equipment impact)
   // 8 = fault (equipment failure)
   // Add one for any unsuppressed alarm that is not acknowledged (for blink).
   70: [CLR(Wrk_Notify) ,GRT(OverTol.Val_Notify,Wrk_Notify) MOV(OverTol.Val_Notify,Wrk_Notify) ,GRT(UnderTol.Val_Notify,Wrk_Notify) MOV(UnderTol.Val_Notify,Wrk_Notify) ,GRT(TareFault.Val_Notify,Wrk_Notify) MOV(TareFault.Val_Notify,Wrk_Notify) ,GRT(EqpFault.Val_Notify,Wrk_Notify) MOV(EqpFault.Val_Notify,Wrk_Notify) ,[XIC(OverTol.Val_Notify.0) ,XIC(UnderTol.Val_Notify.0) ,XIC(TareFault.Val_Notify.0) ,XIC(EqpFault.Val_Notify.0) ] OTE(Wrk_Notify.0) ,MOV(Wrk_Notify,Val_Notify) ];
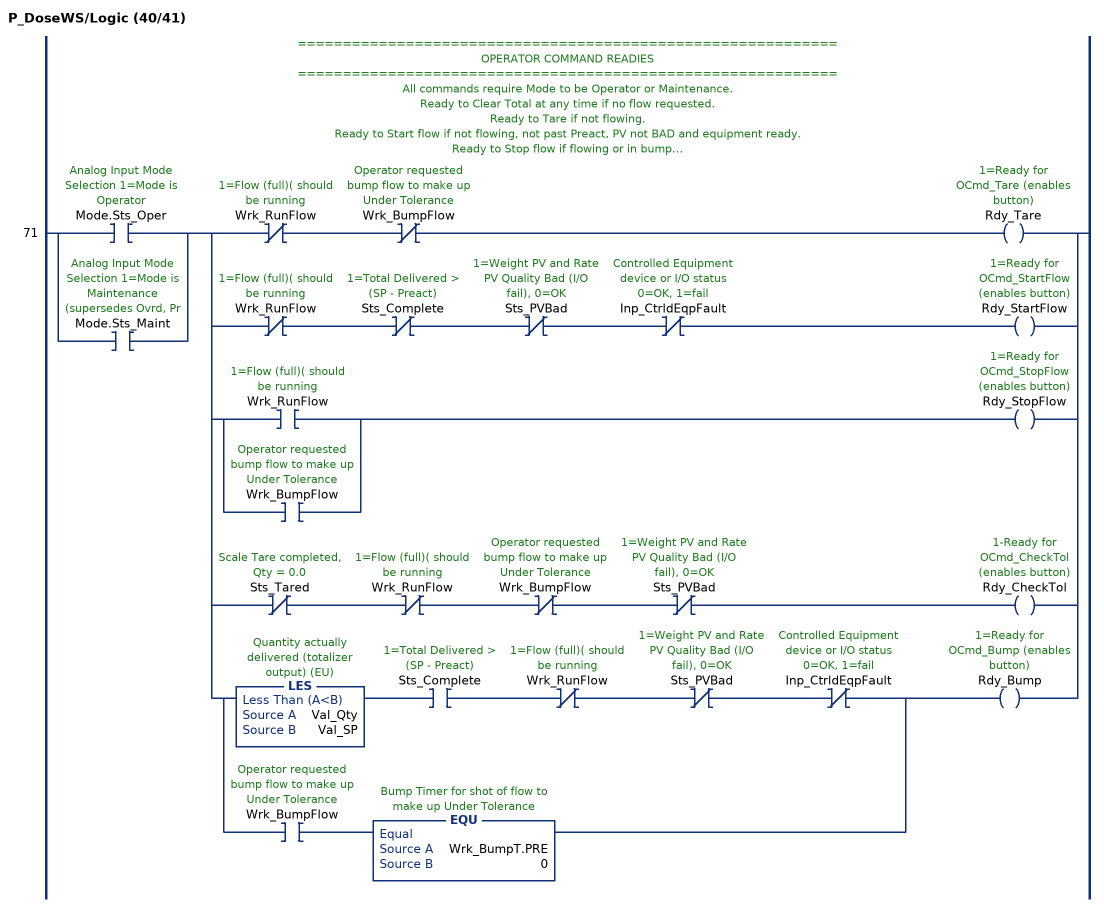
   // ============================================================
   // OPERATOR COMMAND READIES
   // ============================================================
   // All commands require Mode to be Operator or Maintenance.
   // Ready to Clear Total at any time if no flow requested.
   // Ready to Tare if not flowing.
   // Ready to Start flow if not flowing, not past Preact, PV not BAD and equipment ready.
   // Ready to Stop flow if flowing or in bump.
   // Ready to Check Tolerances if PV is not BAD and not flowing.
   // Ready to bump if PV not BAD, past preact but not complete, totalizer is running, and not flowing.
   // NOTE:  Keep the BUMP button active as long as a bump is in progress if
   // the Bump Time is 0 -- this keeps the button on-screen so the bump command is
   // cleared if the operator releases the button!!!
   71: [XIC(Mode.Sts_Oper) ,XIC(Mode.Sts_Maint) ][XIO(Wrk_RunFlow) XIO(Wrk_BumpFlow) OTE(Rdy_Tare) ,XIO(Wrk_RunFlow) XIO(Sts_Complete) XIO(Sts_PVBad) XIO(Inp_CtrldEqpFault) OTE(Rdy_StartFlow) ,[XIC(Wrk_RunFlow) ,XIC(Wrk_BumpFlow) ] OTE(Rdy_StopFlow) ,XIO(Sts_Tared) XIO(Wrk_RunFlow) XIO(Wrk_BumpFlow) XIO(Sts_PVBad) OTE(Rdy_CheckTol) ,[LES(Val_Qty,Val_SP) XIC(Sts_Complete) XIO(Wrk_RunFlow) XIO(Sts_PVBad) XIO(Inp_CtrldEqpFault) ,XIC(Wrk_BumpFlow) EQU(Wrk_BumpT.PRE,0) ] OTE(Rdy_Bump) ];
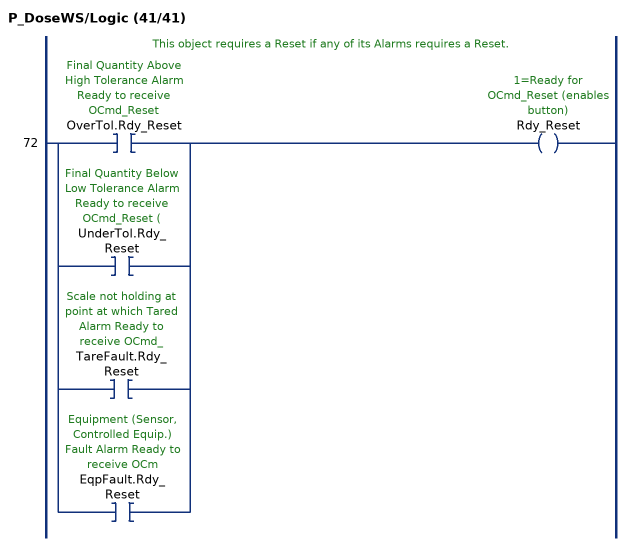
   // This object requires a Reset if any of its Alarms requires a Reset.
   72: [XIC(OverTol.Rdy_Reset) ,XIC(UnderTol.Rdy_Reset) ,XIC(TareFault.Rdy_Reset) ,XIC(EqpFault.Rdy_Reset) ]OTE(Rdy_Reset);
END_ROUTINE
